Fanuc KAREL source: kt00568.KL

-- PROVISIONAL review KL for V770-1; original PC SHA256 2862fa4e773c075f1f902a9a98e6a70591d682fbfeb02a3cc0ba4f09bd7f649a
-- Incomplete behavior may be omitted. Consult companion uncertainty JSON. Do not deploy.
PROGRAM KT00568
%NOLOCKGROUP
VAR
  R2 : REAL
-- UNRESOLVED_DECL V1 type=000013
-- UNRESOLVED_DECL OUT type=000013
BEGIN
  -- UNRESOLVED_PC offsets 5-20; opcodes 2E,22,32,35
  -- UNRESOLVED_PC offsets 25-36; opcodes 2E,23
  -- UNRESOLVED_PC offsets 41-63; opcodes 49,21,8E,4A
  -- UNRESOLVED_PC offsets 68-72; opcodes 7F
END KT00568
